# EPICS autosave request: ip/ipApp/Db/USdigital_T7_settings.req
$(P)USdig_T7:$(S):get_all.SCAN
#$(P)USdig_T7:$(S):A1.DESC
#$(P)USdig_T7:$(S):A1.B
#$(P)USdig_T7:$(S):A2.DESC
#$(P)USdig_T7:$(S):A2.B
$(P)USdig_T7:$(S):Angle.DESC
$(P)USdig_T7:$(S):Angle.B
